# EPICS autosave request: iocBoot/iocoxford/auto_settings.req
file oxford_settings.req P=$(P)
